{attribute 'linkalways'} 
{attribute 'no_explicit_call' := 'This FB is a CLASS and must be accessed using methods or properties'}
{attribute 'enable_dynamic_creation'}
FUNCTION_BLOCK AsyncResponseManager IMPLEMENTS I_AsyncResponseManager
VAR
	sessionStorage : I_SessionStorage;
	responseIdGenerator : I_ResponseIdGenerator;
	headerAccessor : I_AsyncResponseHeaderAccessor;
END_VAR

METHOD ConvertResponseToAsyncResponseSessionData
VAR_INPUT
	Response : I_ServerResponse;
	DestinationAsyncResponse : REFERENCE TO I_AsyncResponseSessionData 
END_VAR
VAR
	sessionId : T_MAXSTRING;
	newResponseId : T_MAXSTRING;
	asyncResponseSessionData : I_AsyncResponseSessionData;
END_VAR
IF NOT headerAccessor.TryGetSessionIdFromResponse(Response,sessionId) THEN
	Response.Error('Unable to create a pending response without a sessionId');
	RETURN;
END_IF

IF ResponseId <> '' THEN
	OriginalResponse.Pending(responseId, RetryDelayInMs);
	RETURN;
END_IF

asyncResponseSessionData := CreateAsyncResponseSessionData(RetryDelayInMs);
newResponseId := responseIdGenerator.Generate();

IF NOT sessionStorage.TryStoreSessionDataById(sessionId, newResponseId, asyncResponseSessionData) THEN
	OriginalResponse.Error('Unable to store pending response');
	asyncResponseSessionData.Dispose();
	RETURN;
END_IF

OriginalResponse.Pending(newResponseId, RetryDelayInMs);
ResponseId := newResponseId;
END_METHOD

METHOD PROTECTED CreateAsyncResponseSessionData : I_AsyncResponseSessionData
VAR_INPUT
	RetryDelayInMs : UDINT;
END_VAR
VAR
	pPendingResponseData : POINTER TO AsyncResponseSessionData;
END_VAR
pPendingResponseData := __NEW(AsyncResponseSessionData(SuggestedRetryDelayInMs := RetryDelayInMs));
CreateAsyncResponseSessionData := pPendingResponseData^;
END_METHOD

METHOD FB_init : BOOL
VAR_INPUT
	bInitRetains : BOOL; // if TRUE, the retain variables are initialized (warm start / cold start)
	bInCopyCode : BOOL;  // if TRUE, the instance afterwards gets moved into the copy code (online change)
	SessionStorage : I_SessionStorage;
	ResponseIdGenerator : I_ResponseIdGenerator;
	HeaderAccessor : I_AsyncResponseHeaderAccessor;
END_VAR
THIS^.sessionStorage := SessionStorage;
THIS^.responseIdGenerator := ResponseIdGenerator;
THIS^.headerAccessor := HeaderAccessor;
END_METHOD

METHOD PUBLIC HandlePending
VAR_INPUT
	OriginalResponse : I_ServerResponse;
	ResponseId : REFERENCE TO T_MAXSTRING;
	RetryDelayInMs : UDINT;
END_VAR
VAR
	sessionId : T_MAXSTRING;
	newResponseId : T_MAXSTRING;
	asyncResponseSessionData : I_AsyncResponseSessionData;
END_VAR
IF NOT headerAccessor.TryGetSessionIdFromResponse(OriginalResponse,sessionId) THEN
	OriginalResponse.Error('Unable to create a pending response without a sessionId');
	RETURN;
END_IF

IF ResponseId <> '' THEN
	OriginalResponse.Pending(responseId, RetryDelayInMs);
	RETURN;
END_IF

asyncResponseSessionData := CreateAsyncResponseSessionData(RetryDelayInMs);
newResponseId := responseIdGenerator.Generate();

IF NOT sessionStorage.TryStoreSessionDataById(sessionId, newResponseId, asyncResponseSessionData) THEN
	OriginalResponse.Error('Unable to store pending response');
	asyncResponseSessionData.Dispose();
	RETURN;
END_IF

OriginalResponse.Pending(newResponseId, RetryDelayInMs);
ResponseId := newResponseId;
END_METHOD

METHOD PUBLIC TryHandleIncomingRequest : BOOL
VAR_INPUT
	Request : I_Request;
	Response : I_ServerResponse;
END_VAR
VAR
	responseId : T_MAXSTRING;
	sessionId : T_MAXSTRING;
	sessionData : I_SessionData;
	asyncResponseData : I_AsyncResponseSessionData;
END_VAR
IF NOT headerAccessor.TryGetResponseIdFromRequest(Request, responseId) THEN
	RETURN;
END_IF

IF NOT headerAccessor.TryGetSessionIdFromRequest(Request, sessionId) THEN
	RETURN;
END_IF

IF NOT sessionStorage.TryRetreiveSessionDataById(sessionId, responseId, sessionData) THEN
	RETURN;
END_IF

IF NOT __QUERYINTERFACE(sessionData, asyncResponseData) THEN
	RETURN;
END_IF

IF asyncResponseData.IsPending THEN
	Response.Pending(responseId, asyncResponseData.SuggestedRetryDelayInMs);
	TryHandleIncomingRequest := TRUE;
	RETURN;
END_IF

IF NOT asyncResponseData.TryUpdateServerResponse(Response) THEN	
	Response.Error('Unable to update server response with pending data');
	TryHandleIncomingRequest := TRUE;
	RETURN;
END_IF

sessionStorage.DisposeSessionDataById(sessionId, responseId);
TryHandleIncomingRequest := TRUE;
END_METHOD

END_FUNCTION_BLOCK

(* stored: Version 1.1.0.1, ProductVersion 3.1.4024.12
   POU AsyncResponseManager: Id {227d2639-d4f9-47c2-ab56-861a5448ae71}, SpecialFunc None
   Folder Constructor: Id {512c79a0-d7ea-4632-8454-ff0bdda61950}
   Folder Protected: Id {10f5e310-740f-44f6-88d4-6719d1d292b2}
   Method ConvertResponseToAsyncResponseSessionData: Id {9b1dd38d-7371-4b2c-aeed-2ce787286b24}
   Method CreateAsyncResponseSessionData: Id {9309a56c-b4a3-406f-ba56-d711c30ffecf}
   Method FB_init: Id {10c5352a-129b-4eaa-abe3-146411036763}
   Method HandlePending: Id {fab2cba9-29a7-40ae-840c-2912fb9461bb}
   Method TryHandleIncomingRequest: Id {5dd32684-e554-429c-8b1d-ad94c31a0043} *)
